FUNCTION_BLOCK Test_F_DateTimeAsString_ReturnsDateTimeString EXTENDS TUnitTestBase
VAR
    TimeStruct : TIMESTRUCT := (wDay := 23, wMonth := 12, wYear := 1945, wHour := 22, wMinute := 20, wSecond := 18);
END_VAR

Assertion.AssertEquals_STRING(
    Expected := '22:20:18 23/12/1945',
    Actual   := F_DateTimeAsString(TimeStruct),
    ObjectName := _TestName,
    VariableName  := 'F_DateTimeAsString(TimeStruct)');


TestFinished();

END_FUNCTION_BLOCK

(* stored: Version 1.1.0.1, ProductVersion 3.1.4024.4
   POU Test_F_DateTimeAsString_ReturnsDateTimeString: Id {70721f54-ad56-0ed4-217d-cb50130dc051}, SpecialFunc None *)
